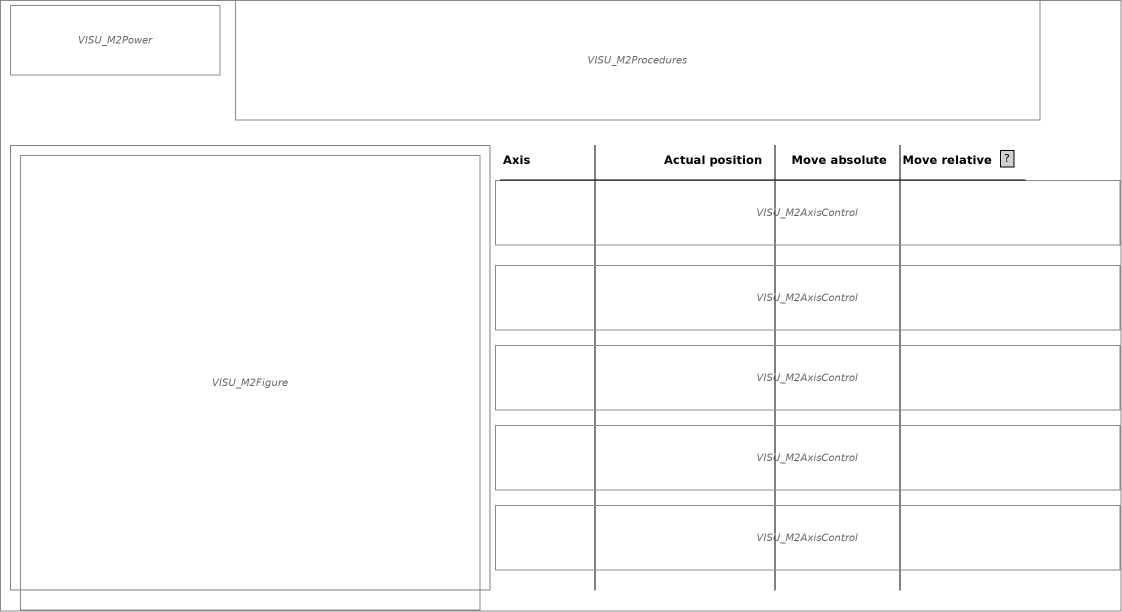
VISUALIZATION VISU_M2Axes  // 1122x612
VAR_IN_OUT
	ref : M2;
    widget : M2Widget;
END_VAR
    Line (595,590) (595,145)
    Line (775,590) (775,145)
    Line (900,590) (900,145)
    Rectangle (10,145 480x445)
    Frame (20,155 460x455)
        shows VISU_M2Figure(ref := ref, widget := widget.figure)
    Frame (10,5 210x70)
        shows VISU_M2Power(ref := ref, widget := widget)
    Frame (495,180 625x65)
        shows VISU_M2AxisControl(widget := widget.x)
    Frame (495,265 625x65)
        shows VISU_M2AxisControl(widget := widget.y)
    Frame (495,345 625x65)
        shows VISU_M2AxisControl(widget := widget.z)
    Frame (495,425 625x65)
        shows VISU_M2AxisControl(widget := widget.tiltX)
    Frame (495,505 625x65)
        shows VISU_M2AxisControl(widget := widget.tiltY)
    Line (1025,180) (500,180)
    Label (500,145 95x30), "Axis"
    Label (605,145 160x30), "Actual position"
    Label (780,145 110x30), "Move absolute"
    Label (900,145 95x30), "Move relative"
    Frame (235,0 805x120)
        shows VISU_M2Procedures(ref := ref, widget := widget)
    RoundedRectangle (1000,150 14x17), "?", tooltip "Faster (<<< or >>>) in the direction without backlash"
END_VISUALIZATION

(* stored: Version 1.1.0.1, ProductVersion 3.1.4019.2
   Visu VISU_M2Axes: Id {fd214743-8b45-4df1-b196-781b5a1325e9} *)
